// TIA Portal V15.1 export
// export: Created 2024-05-17T05:38:57.384126Z, ExportSetting WithDefaults, DisplayName Totally Integrated Automation Portal, DisplayVersion V15.1 Update 5, DisplayName TIA Portal Openness, DisplayVersion V15.1 Update 5, DisplayName SINAMICS Startdrive Advanced, DisplayVersion V15.1, DisplayName G130, G150, S120, S150, SINAMICS MV, S210, DisplayVersion V15.1, DisplayName G110M, G120, G120C, G120D, G120P, DisplayVersion V15.1, DisplayName STEP 7 Professional, DisplayVersion V15.1 Update 5, DisplayName STEP 7 Safety, DisplayVersion V15.1, DisplayName WinCC Professional, DisplayVersion V15.1 Update 5, DisplayName SIMATIC Visualization Architect, DisplayVersion V15.1
FUNCTION "209210ZS01Safety" : Void   // FC325, FBD
TITLE = 209210ZS01 Safety
{ S7_Optimized_Access := 'FALSE' }
AUTHOR : VCG
FAMILY : Local
NAME : 610
VERSION : 0.1
// stored: AutoNumber false, IsIECCheckEnabled false, SetENOAutomatically False, UDAEnableTagReadback false
   VAR_OUTPUT
      O_AlarmA : Bool;   // Alarm A
      O_AlarmB : Bool;   // Alarm B
      O_AlarmC : Bool;   // Alarm C
      O_AlarmD : Bool;   // Alarm D
      O_AlarmABCondition : Bool;   // Alarms resetable
      H_IAnim : Word;   // Icon Animation
   END_VAR
BEGIN

REGION Network 1: **** 2.1 - Enable Alarms **** 210CS22M4SG10F & SG11F Check if both safety sensors are activated
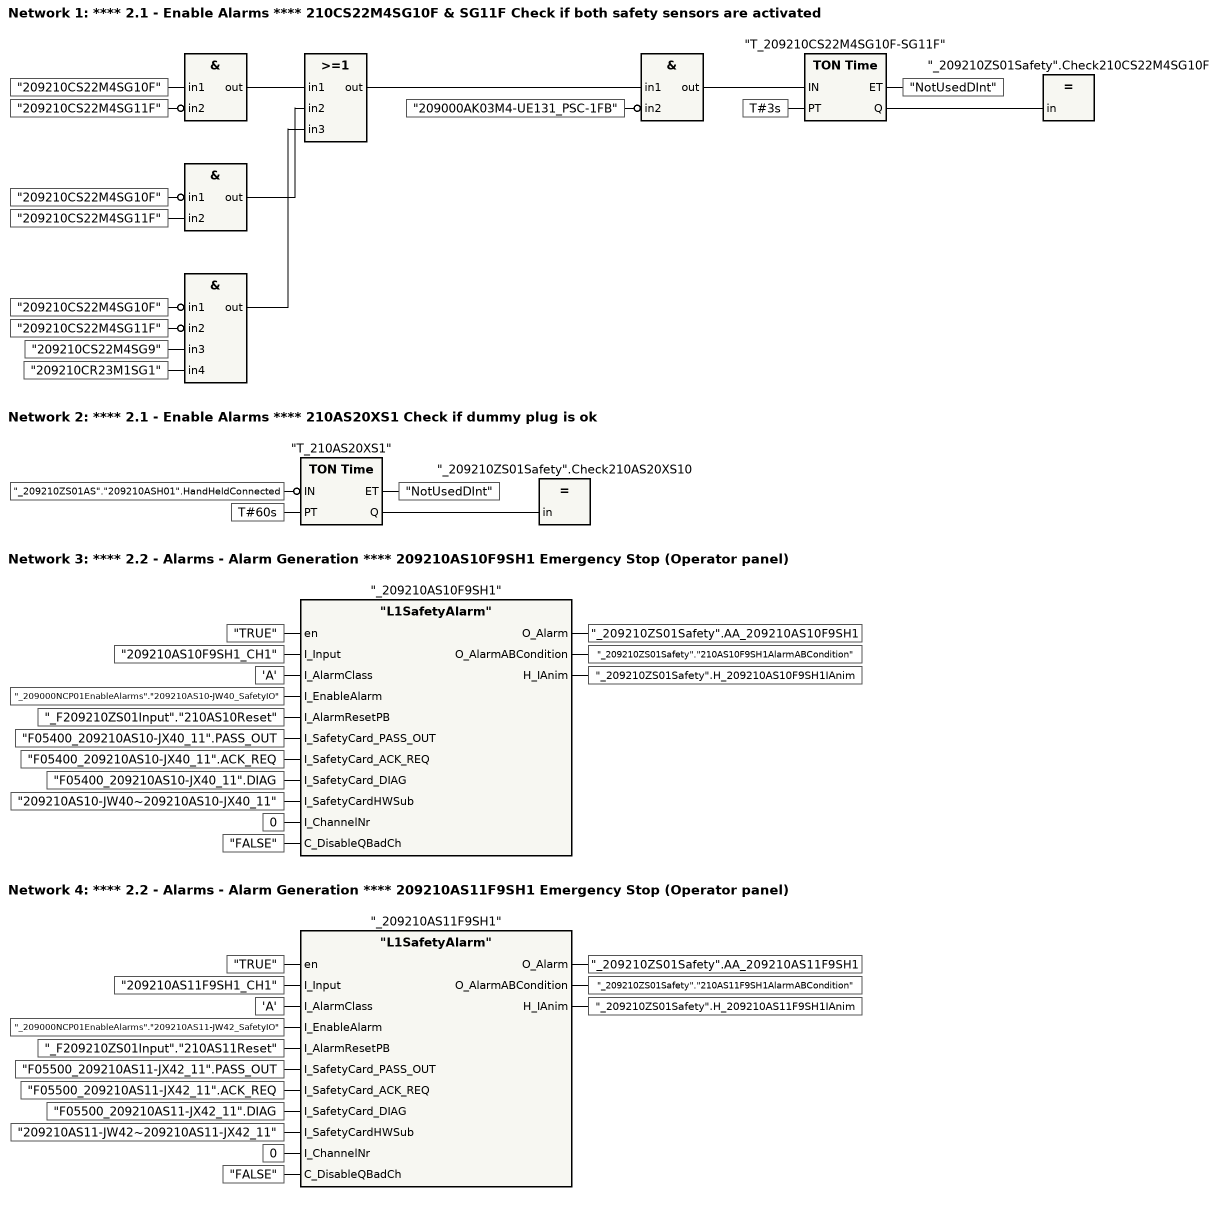
   "T_209210CS22M4SG10F-SG11F".TON(IN := (("209210CS22M4SG10F" AND NOT "209210CS22M4SG11F") OR (NOT "209210CS22M4SG10F" AND "209210CS22M4SG11F") OR (NOT "209210CS22M4SG10F" AND NOT "209210CS22M4SG11F" AND "209210CS22M4SG9" AND "209210CR23M1SG1")) AND NOT "209000AK03M4-UE131_PSC-1FB",
                           PT := T#3s,
                           ET => "NotUsedDInt");
   "_209210ZS01Safety".Check210CS22M4SG10F := "T_209210CS22M4SG10F-SG11F".Q;
END_REGION

REGION Network 2: **** 2.1 - Enable Alarms **** 210AS20XS1 Check if dummy plug is ok
   "T_210AS20XS1".TON(IN := NOT "_209210ZS01AS"."209210ASH01".HandHeldConnected,
                      PT := T#60s,
                      ET => "NotUsedDInt");
   "_209210ZS01Safety".Check210AS20XS10 := "T_210AS20XS1".Q;
END_REGION

REGION Network 3: **** 2.2 - Alarms - Alarm Generation **** 209210AS10F9SH1 Emergency Stop (Operator panel)
   // Emergency Stop
   IF "TRUE" THEN
       "_209210AS10F9SH1"(I_Input := "209210AS10F9SH1_CH1",   // "L1SafetyAlarm"
                          I_AlarmClass := 'A',
                          I_EnableAlarm := "_209000NCP01EnableAlarms"."209210AS10-JW40_SafetyIO",
                          I_AlarmResetPB := "_F209210ZS01Input"."210AS10Reset",
                          I_SafetyCard_PASS_OUT := "F05400_209210AS10-JX40_11".PASS_OUT,
                          I_SafetyCard_ACK_REQ := "F05400_209210AS10-JX40_11".ACK_REQ,
                          I_SafetyCard_DIAG := "F05400_209210AS10-JX40_11".DIAG,
                          I_SafetyCardHWSub := "209210AS10-JW40~209210AS10-JX40_11",
                          I_ChannelNr := 0,
                          C_DisableQBadCh := "FALSE",
                          O_Alarm => "_209210ZS01Safety".AA_209210AS10F9SH1,
                          O_AlarmABCondition => "_209210ZS01Safety"."210AS10F9SH1AlarmABCondition",
                          H_IAnim => "_209210ZS01Safety".H_209210AS10F9SH1IAnim);
   END_IF;
END_REGION

REGION Network 4: **** 2.2 - Alarms - Alarm Generation **** 209210AS11F9SH1 Emergency Stop (Operator panel)
   // Emergency Stop
   IF "TRUE" THEN
       "_209210AS11F9SH1"(I_Input := "209210AS11F9SH1_CH1",   // "L1SafetyAlarm"
                          I_AlarmClass := 'A',
                          I_EnableAlarm := "_209000NCP01EnableAlarms"."209210AS11-JW42_SafetyIO",
                          I_AlarmResetPB := "_F209210ZS01Input"."210AS11Reset",
                          I_SafetyCard_PASS_OUT := "F05500_209210AS11-JX42_11".PASS_OUT,
                          I_SafetyCard_ACK_REQ := "F05500_209210AS11-JX42_11".ACK_REQ,
                          I_SafetyCard_DIAG := "F05500_209210AS11-JX42_11".DIAG,
                          I_SafetyCardHWSub := "209210AS11-JW42~209210AS11-JX42_11",
                          I_ChannelNr := 0,
                          C_DisableQBadCh := "FALSE",
                          O_Alarm => "_209210ZS01Safety".AA_209210AS11F9SH1,
                          O_AlarmABCondition => "_209210ZS01Safety"."210AS11F9SH1AlarmABCondition",
                          H_IAnim => "_209210ZS01Safety".H_209210AS11F9SH1IAnim);
   END_IF;
END_REGION

REGION Network 5: **** 2.2 - Alarms - Alarm Generation **** 209210AS20F9SH1 Emergency Stop (Start/Stop panel)
   // Emergency Stop
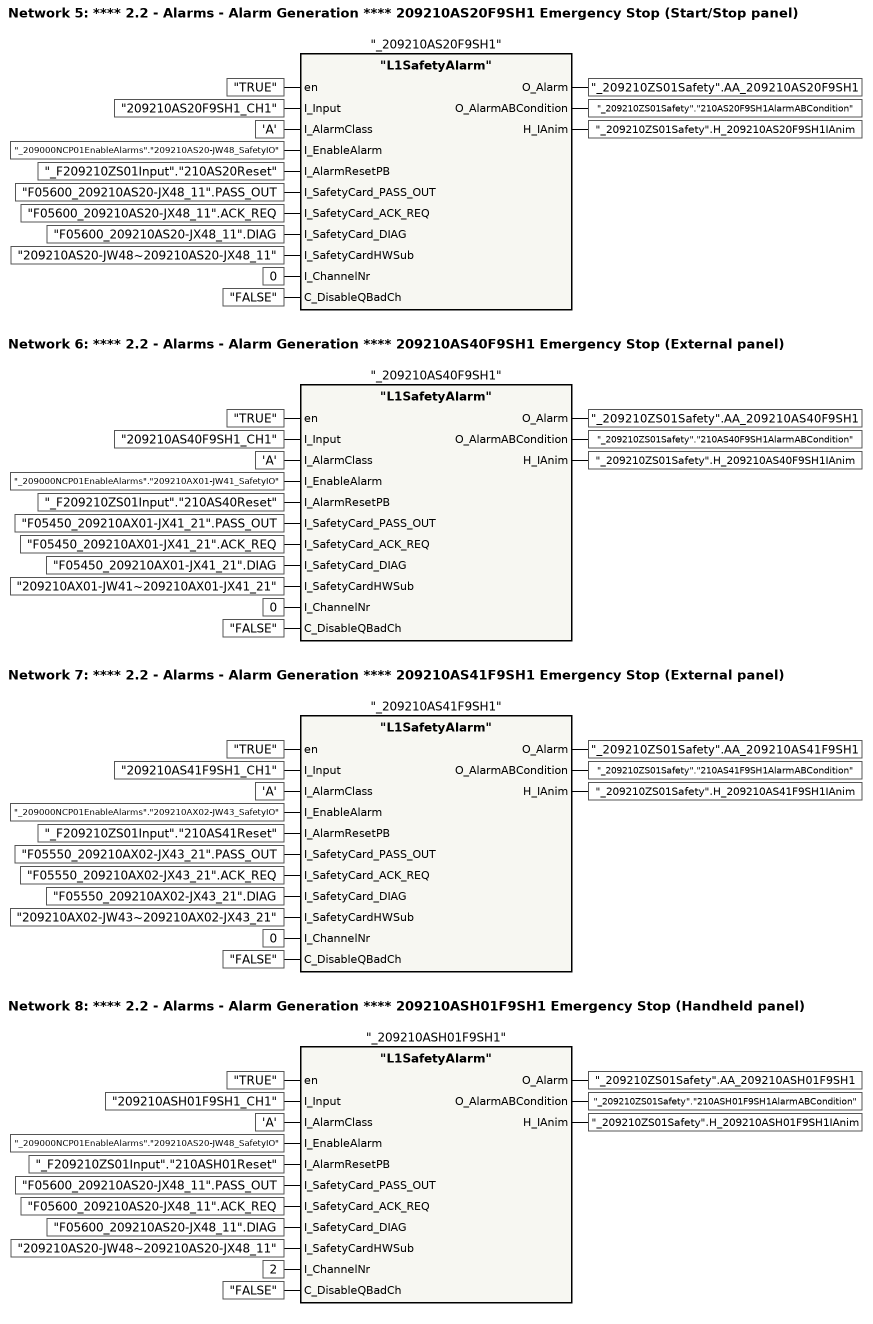
   IF "TRUE" THEN
       "_209210AS20F9SH1"(I_Input := "209210AS20F9SH1_CH1",   // "L1SafetyAlarm"
                          I_AlarmClass := 'A',
                          I_EnableAlarm := "_209000NCP01EnableAlarms"."209210AS20-JW48_SafetyIO",
                          I_AlarmResetPB := "_F209210ZS01Input"."210AS20Reset",
                          I_SafetyCard_PASS_OUT := "F05600_209210AS20-JX48_11".PASS_OUT,
                          I_SafetyCard_ACK_REQ := "F05600_209210AS20-JX48_11".ACK_REQ,
                          I_SafetyCard_DIAG := "F05600_209210AS20-JX48_11".DIAG,
                          I_SafetyCardHWSub := "209210AS20-JW48~209210AS20-JX48_11",
                          I_ChannelNr := 0,
                          C_DisableQBadCh := "FALSE",
                          O_Alarm => "_209210ZS01Safety".AA_209210AS20F9SH1,
                          O_AlarmABCondition => "_209210ZS01Safety"."210AS20F9SH1AlarmABCondition",
                          H_IAnim => "_209210ZS01Safety".H_209210AS20F9SH1IAnim);
   END_IF;
END_REGION

REGION Network 6: **** 2.2 - Alarms - Alarm Generation **** 209210AS40F9SH1 Emergency Stop (External panel)
   // Emergency Stop
   IF "TRUE" THEN
       "_209210AS40F9SH1"(I_Input := "209210AS40F9SH1_CH1",   // "L1SafetyAlarm"
                          I_AlarmClass := 'A',
                          I_EnableAlarm := "_209000NCP01EnableAlarms"."209210AX01-JW41_SafetyIO",
                          I_AlarmResetPB := "_F209210ZS01Input"."210AS40Reset",
                          I_SafetyCard_PASS_OUT := "F05450_209210AX01-JX41_21".PASS_OUT,
                          I_SafetyCard_ACK_REQ := "F05450_209210AX01-JX41_21".ACK_REQ,
                          I_SafetyCard_DIAG := "F05450_209210AX01-JX41_21".DIAG,
                          I_SafetyCardHWSub := "209210AX01-JW41~209210AX01-JX41_21",
                          I_ChannelNr := 0,
                          C_DisableQBadCh := "FALSE",
                          O_Alarm => "_209210ZS01Safety".AA_209210AS40F9SH1,
                          O_AlarmABCondition => "_209210ZS01Safety"."210AS40F9SH1AlarmABCondition",
                          H_IAnim => "_209210ZS01Safety".H_209210AS40F9SH1IAnim);
   END_IF;
END_REGION

REGION Network 7: **** 2.2 - Alarms - Alarm Generation **** 209210AS41F9SH1 Emergency Stop (External panel)
   // Emergency Stop
   IF "TRUE" THEN
       "_209210AS41F9SH1"(I_Input := "209210AS41F9SH1_CH1",   // "L1SafetyAlarm"
                          I_AlarmClass := 'A',
                          I_EnableAlarm := "_209000NCP01EnableAlarms"."209210AX02-JW43_SafetyIO",
                          I_AlarmResetPB := "_F209210ZS01Input"."210AS41Reset",
                          I_SafetyCard_PASS_OUT := "F05550_209210AX02-JX43_21".PASS_OUT,
                          I_SafetyCard_ACK_REQ := "F05550_209210AX02-JX43_21".ACK_REQ,
                          I_SafetyCard_DIAG := "F05550_209210AX02-JX43_21".DIAG,
                          I_SafetyCardHWSub := "209210AX02-JW43~209210AX02-JX43_21",
                          I_ChannelNr := 0,
                          C_DisableQBadCh := "FALSE",
                          O_Alarm => "_209210ZS01Safety".AA_209210AS41F9SH1,
                          O_AlarmABCondition => "_209210ZS01Safety"."210AS41F9SH1AlarmABCondition",
                          H_IAnim => "_209210ZS01Safety".H_209210AS41F9SH1IAnim);
   END_IF;
END_REGION

REGION Network 8: **** 2.2 - Alarms - Alarm Generation **** 209210ASH01F9SH1 Emergency Stop (Handheld panel)
   // Emergency Stop
   IF "TRUE" THEN
       "_209210ASH01F9SH1"(I_Input := "209210ASH01F9SH1_CH1",   // "L1SafetyAlarm"
                           I_AlarmClass := 'A',
                           I_EnableAlarm := "_209000NCP01EnableAlarms"."209210AS20-JW48_SafetyIO",
                           I_AlarmResetPB := "_F209210ZS01Input"."210ASH01Reset",
                           I_SafetyCard_PASS_OUT := "F05600_209210AS20-JX48_11".PASS_OUT,
                           I_SafetyCard_ACK_REQ := "F05600_209210AS20-JX48_11".ACK_REQ,
                           I_SafetyCard_DIAG := "F05600_209210AS20-JX48_11".DIAG,
                           I_SafetyCardHWSub := "209210AS20-JW48~209210AS20-JX48_11",
                           I_ChannelNr := 2,
                           C_DisableQBadCh := "FALSE",
                           O_Alarm => "_209210ZS01Safety".AA_209210ASH01F9SH1,
                           O_AlarmABCondition => "_209210ZS01Safety"."210ASH01F9SH1AlarmABCondition",
                           H_IAnim => "_209210ZS01Safety".H_209210ASH01F9SH1IAnim);
   END_IF;
END_REGION

REGION Network 9: **** 2.2 - Alarms - Alarm Generation **** 209210ASH01F9SH2 Deathmans switch (Handheld panel)
   // Deathmans switch
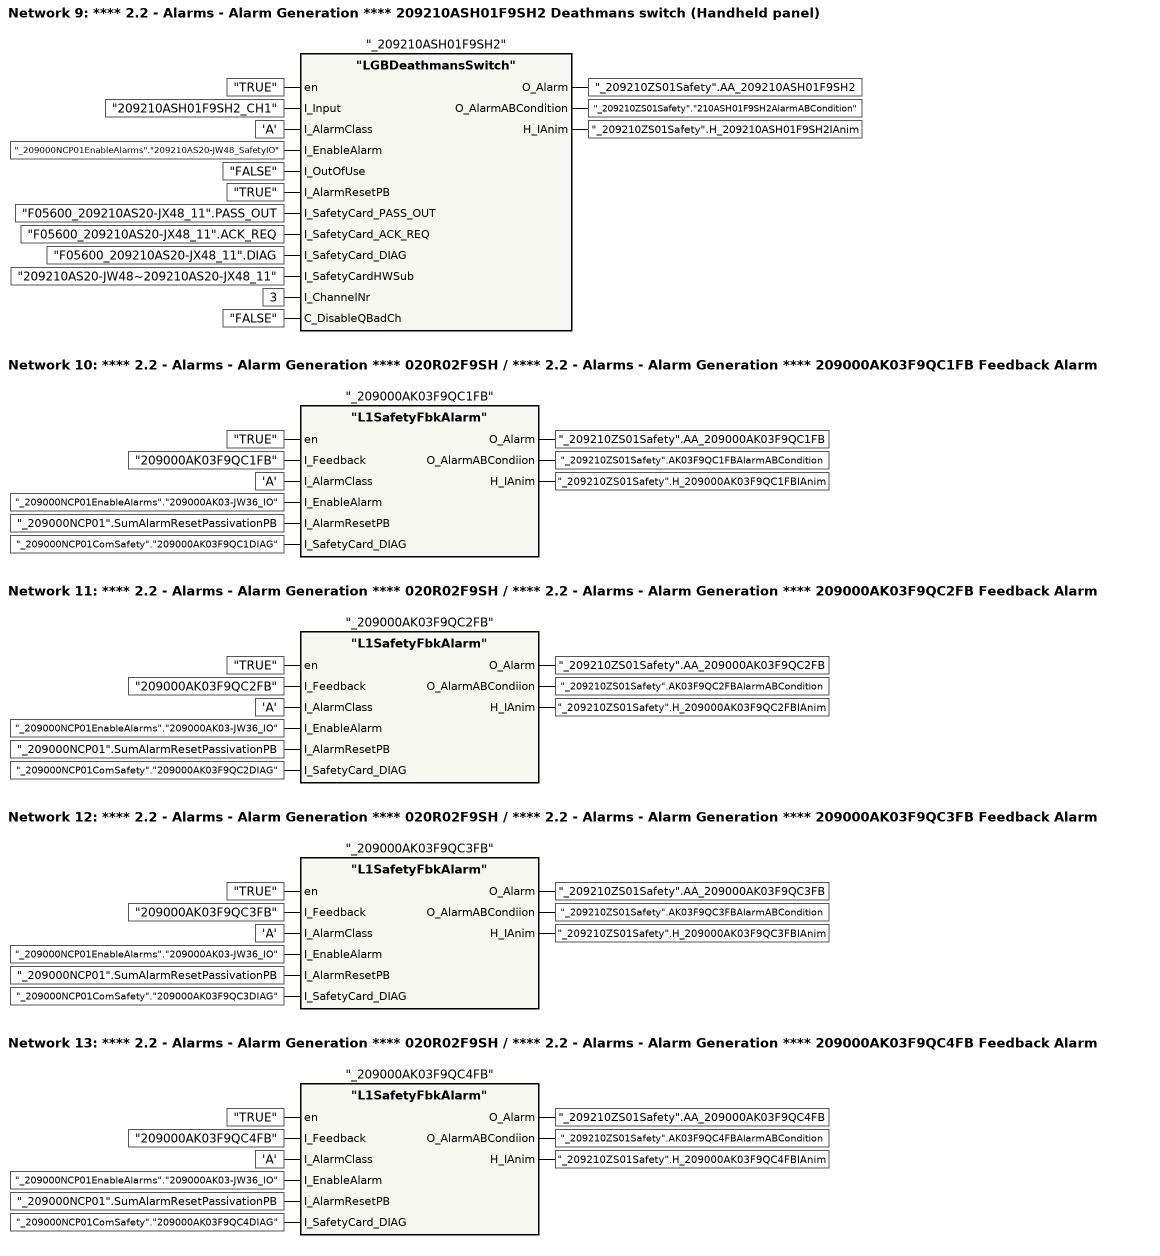
   IF "TRUE" THEN
       "_209210ASH01F9SH2"(I_Input := "209210ASH01F9SH2_CH1",   // "LGBDeathmansSwitch"
                           I_AlarmClass := 'A',
                           I_EnableAlarm := "_209000NCP01EnableAlarms"."209210AS20-JW48_SafetyIO",
                           I_OutOfUse := "FALSE",
                           I_AlarmResetPB := "TRUE",
                           I_SafetyCard_PASS_OUT := "F05600_209210AS20-JX48_11".PASS_OUT,
                           I_SafetyCard_ACK_REQ := "F05600_209210AS20-JX48_11".ACK_REQ,
                           I_SafetyCard_DIAG := "F05600_209210AS20-JX48_11".DIAG,
                           I_SafetyCardHWSub := "209210AS20-JW48~209210AS20-JX48_11",
                           I_ChannelNr := 3,
                           C_DisableQBadCh := "FALSE",
                           O_Alarm => "_209210ZS01Safety".AA_209210ASH01F9SH2,
                           O_AlarmABCondition => "_209210ZS01Safety"."210ASH01F9SH2AlarmABCondition",
                           H_IAnim => "_209210ZS01Safety".H_209210ASH01F9SH2IAnim);
   END_IF;
END_REGION

REGION Network 10: **** 2.2 - Alarms - Alarm Generation **** 020R02F9SH / **** 2.2 - Alarms - Alarm Generation **** 209000AK03F9QC1FB Feedback Alarm
   // E-Stop Push Button / Feedback Alarm
   IF "TRUE" THEN
       "_209000AK03F9QC1FB"(I_Feedback := "209000AK03F9QC1FB",   // "L1SafetyFbkAlarm"
                            I_AlarmClass := 'A',
                            I_EnableAlarm := "_209000NCP01EnableAlarms"."209000AK03-JW36_IO",
                            I_AlarmResetPB := "_209000NCP01".SumAlarmResetPassivationPB,
                            I_SafetyCard_DIAG := "_209000NCP01ComSafety"."209000AK03F9QC1DIAG",
                            O_Alarm => "_209210ZS01Safety".AA_209000AK03F9QC1FB,
                            O_AlarmABCondiion => "_209210ZS01Safety".AK03F9QC1FBAlarmABCondition,
                            H_IAnim => "_209210ZS01Safety".H_209000AK03F9QC1FBIAnim);
   END_IF;
END_REGION

REGION Network 11: **** 2.2 - Alarms - Alarm Generation **** 020R02F9SH / **** 2.2 - Alarms - Alarm Generation **** 209000AK03F9QC2FB Feedback Alarm
   // E-Stop Push Button / Feedback Alarm
   IF "TRUE" THEN
       "_209000AK03F9QC2FB"(I_Feedback := "209000AK03F9QC2FB",   // "L1SafetyFbkAlarm"
                            I_AlarmClass := 'A',
                            I_EnableAlarm := "_209000NCP01EnableAlarms"."209000AK03-JW36_IO",
                            I_AlarmResetPB := "_209000NCP01".SumAlarmResetPassivationPB,
                            I_SafetyCard_DIAG := "_209000NCP01ComSafety"."209000AK03F9QC2DIAG",
                            O_Alarm => "_209210ZS01Safety".AA_209000AK03F9QC2FB,
                            O_AlarmABCondiion => "_209210ZS01Safety".AK03F9QC2FBAlarmABCondition,
                            H_IAnim => "_209210ZS01Safety".H_209000AK03F9QC2FBIAnim);
   END_IF;
END_REGION

REGION Network 12: **** 2.2 - Alarms - Alarm Generation **** 020R02F9SH / **** 2.2 - Alarms - Alarm Generation **** 209000AK03F9QC3FB Feedback Alarm
   // E-Stop Push Button / Feedback Alarm
   IF "TRUE" THEN
       "_209000AK03F9QC3FB"(I_Feedback := "209000AK03F9QC3FB",   // "L1SafetyFbkAlarm"
                            I_AlarmClass := 'A',
                            I_EnableAlarm := "_209000NCP01EnableAlarms"."209000AK03-JW36_IO",
                            I_AlarmResetPB := "_209000NCP01".SumAlarmResetPassivationPB,
                            I_SafetyCard_DIAG := "_209000NCP01ComSafety"."209000AK03F9QC3DIAG",
                            O_Alarm => "_209210ZS01Safety".AA_209000AK03F9QC3FB,
                            O_AlarmABCondiion => "_209210ZS01Safety".AK03F9QC3FBAlarmABCondition,
                            H_IAnim => "_209210ZS01Safety".H_209000AK03F9QC3FBIAnim);
   END_IF;
END_REGION

REGION Network 13: **** 2.2 - Alarms - Alarm Generation **** 020R02F9SH / **** 2.2 - Alarms - Alarm Generation **** 209000AK03F9QC4FB Feedback Alarm
   // E-Stop Push Button / Feedback Alarm
   IF "TRUE" THEN
       "_209000AK03F9QC4FB"(I_Feedback := "209000AK03F9QC4FB",   // "L1SafetyFbkAlarm"
                            I_AlarmClass := 'A',
                            I_EnableAlarm := "_209000NCP01EnableAlarms"."209000AK03-JW36_IO",
                            I_AlarmResetPB := "_209000NCP01".SumAlarmResetPassivationPB,
                            I_SafetyCard_DIAG := "_209000NCP01ComSafety"."209000AK03F9QC4DIAG",
                            O_Alarm => "_209210ZS01Safety".AA_209000AK03F9QC4FB,
                            O_AlarmABCondiion => "_209210ZS01Safety".AK03F9QC4FBAlarmABCondition,
                            H_IAnim => "_209210ZS01Safety".H_209000AK03F9QC4FBIAnim);
   END_IF;
END_REGION

REGION Network 14: **** 2.2 - Alarms - Alarm Generation **** 020R02F9SH / **** 2.2 - Alarms - Alarm Generation **** 209000AK03F9QC5FB Feedback Alarm
   // E-Stop Push Button / Feedback Alarm
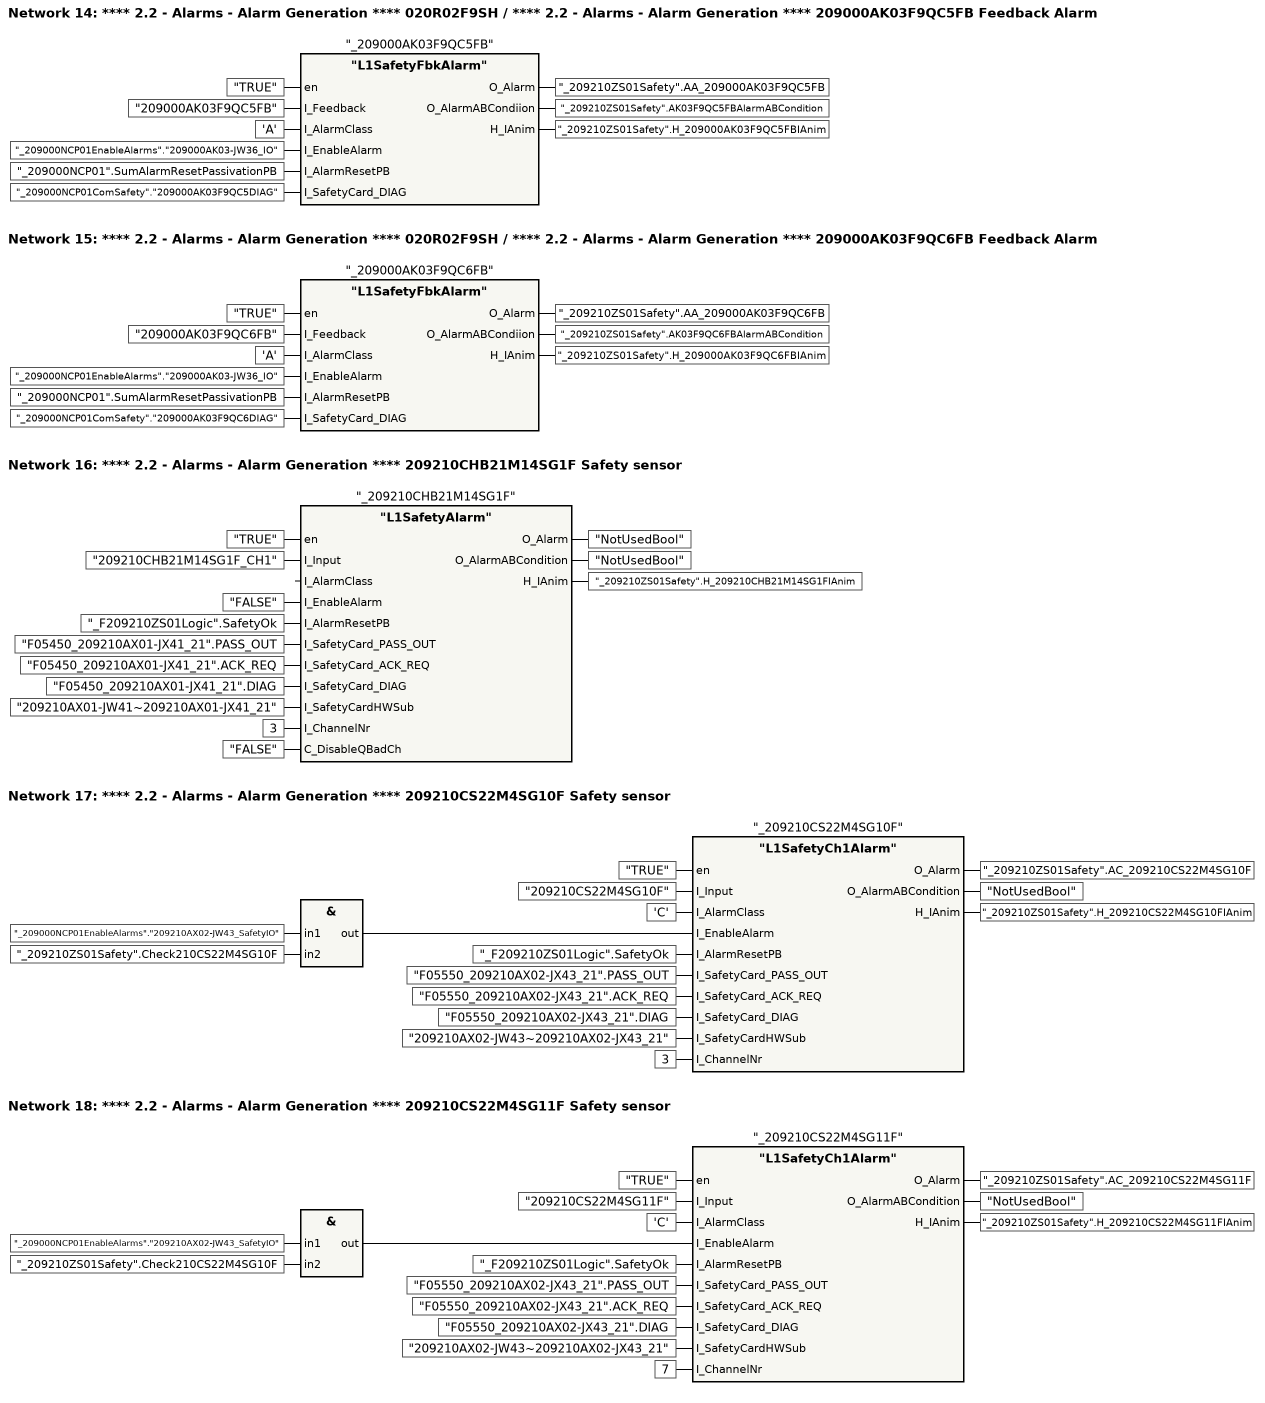
   IF "TRUE" THEN
       "_209000AK03F9QC5FB"(I_Feedback := "209000AK03F9QC5FB",   // "L1SafetyFbkAlarm"
                            I_AlarmClass := 'A',
                            I_EnableAlarm := "_209000NCP01EnableAlarms"."209000AK03-JW36_IO",
                            I_AlarmResetPB := "_209000NCP01".SumAlarmResetPassivationPB,
                            I_SafetyCard_DIAG := "_209000NCP01ComSafety"."209000AK03F9QC5DIAG",
                            O_Alarm => "_209210ZS01Safety".AA_209000AK03F9QC5FB,
                            O_AlarmABCondiion => "_209210ZS01Safety".AK03F9QC5FBAlarmABCondition,
                            H_IAnim => "_209210ZS01Safety".H_209000AK03F9QC5FBIAnim);
   END_IF;
END_REGION

REGION Network 15: **** 2.2 - Alarms - Alarm Generation **** 020R02F9SH / **** 2.2 - Alarms - Alarm Generation **** 209000AK03F9QC6FB Feedback Alarm
   // E-Stop Push Button / Feedback Alarm
   IF "TRUE" THEN
       "_209000AK03F9QC6FB"(I_Feedback := "209000AK03F9QC6FB",   // "L1SafetyFbkAlarm"
                            I_AlarmClass := 'A',
                            I_EnableAlarm := "_209000NCP01EnableAlarms"."209000AK03-JW36_IO",
                            I_AlarmResetPB := "_209000NCP01".SumAlarmResetPassivationPB,
                            I_SafetyCard_DIAG := "_209000NCP01ComSafety"."209000AK03F9QC6DIAG",
                            O_Alarm => "_209210ZS01Safety".AA_209000AK03F9QC6FB,
                            O_AlarmABCondiion => "_209210ZS01Safety".AK03F9QC6FBAlarmABCondition,
                            H_IAnim => "_209210ZS01Safety".H_209000AK03F9QC6FBIAnim);
   END_IF;
END_REGION

REGION Network 16: **** 2.2 - Alarms - Alarm Generation **** 209210CHB21M14SG1F Safety sensor
   // Safety sensor
   IF "TRUE" THEN
       "_209210CHB21M14SG1F"(I_Input := "209210CHB21M14SG1F_CH1",   // "L1SafetyAlarm"
                             I_EnableAlarm := "FALSE",
                             I_AlarmResetPB := "_F209210ZS01Logic".SafetyOk,
                             I_SafetyCard_PASS_OUT := "F05450_209210AX01-JX41_21".PASS_OUT,
                             I_SafetyCard_ACK_REQ := "F05450_209210AX01-JX41_21".ACK_REQ,
                             I_SafetyCard_DIAG := "F05450_209210AX01-JX41_21".DIAG,
                             I_SafetyCardHWSub := "209210AX01-JW41~209210AX01-JX41_21",
                             I_ChannelNr := 3,
                             C_DisableQBadCh := "FALSE",
                             O_Alarm => "NotUsedBool",
                             O_AlarmABCondition => "NotUsedBool",
                             H_IAnim => "_209210ZS01Safety".H_209210CHB21M14SG1FIAnim);
   END_IF;
END_REGION

REGION Network 17: **** 2.2 - Alarms - Alarm Generation **** 209210CS22M4SG10F Safety sensor
   // Safety sensor
   IF "TRUE" THEN
       "_209210CS22M4SG10F"(I_Input := "209210CS22M4SG10F",   // "L1SafetyCh1Alarm"
                            I_AlarmClass := 'C',
                            I_EnableAlarm := "_209000NCP01EnableAlarms"."209210AX02-JW43_SafetyIO" AND "_209210ZS01Safety".Check210CS22M4SG10F,
                            I_AlarmResetPB := "_F209210ZS01Logic".SafetyOk,
                            I_SafetyCard_PASS_OUT := "F05550_209210AX02-JX43_21".PASS_OUT,
                            I_SafetyCard_ACK_REQ := "F05550_209210AX02-JX43_21".ACK_REQ,
                            I_SafetyCard_DIAG := "F05550_209210AX02-JX43_21".DIAG,
                            I_SafetyCardHWSub := "209210AX02-JW43~209210AX02-JX43_21",
                            I_ChannelNr := 3,
                            O_Alarm => "_209210ZS01Safety".AC_209210CS22M4SG10F,
                            O_AlarmABCondition => "NotUsedBool",
                            H_IAnim => "_209210ZS01Safety".H_209210CS22M4SG10FIAnim);
   END_IF;
END_REGION

REGION Network 18: **** 2.2 - Alarms - Alarm Generation **** 209210CS22M4SG11F Safety sensor
   // Safety sensor
   IF "TRUE" THEN
       "_209210CS22M4SG11F"(I_Input := "209210CS22M4SG11F",   // "L1SafetyCh1Alarm"
                            I_AlarmClass := 'C',
                            I_EnableAlarm := "_209000NCP01EnableAlarms"."209210AX02-JW43_SafetyIO" AND "_209210ZS01Safety".Check210CS22M4SG10F,
                            I_AlarmResetPB := "_F209210ZS01Logic".SafetyOk,
                            I_SafetyCard_PASS_OUT := "F05550_209210AX02-JX43_21".PASS_OUT,
                            I_SafetyCard_ACK_REQ := "F05550_209210AX02-JX43_21".ACK_REQ,
                            I_SafetyCard_DIAG := "F05550_209210AX02-JX43_21".DIAG,
                            I_SafetyCardHWSub := "209210AX02-JW43~209210AX02-JX43_21",
                            I_ChannelNr := 7,
                            O_Alarm => "_209210ZS01Safety".AC_209210CS22M4SG11F,
                            O_AlarmABCondition => "NotUsedBool",
                            H_IAnim => "_209210ZS01Safety".H_209210CS22M4SG11FIAnim);
   END_IF;
END_REGION

REGION Network 19: **** 2.2 - Alarms - Alarm Generation **** 209210AS20XS10 Dummy plug
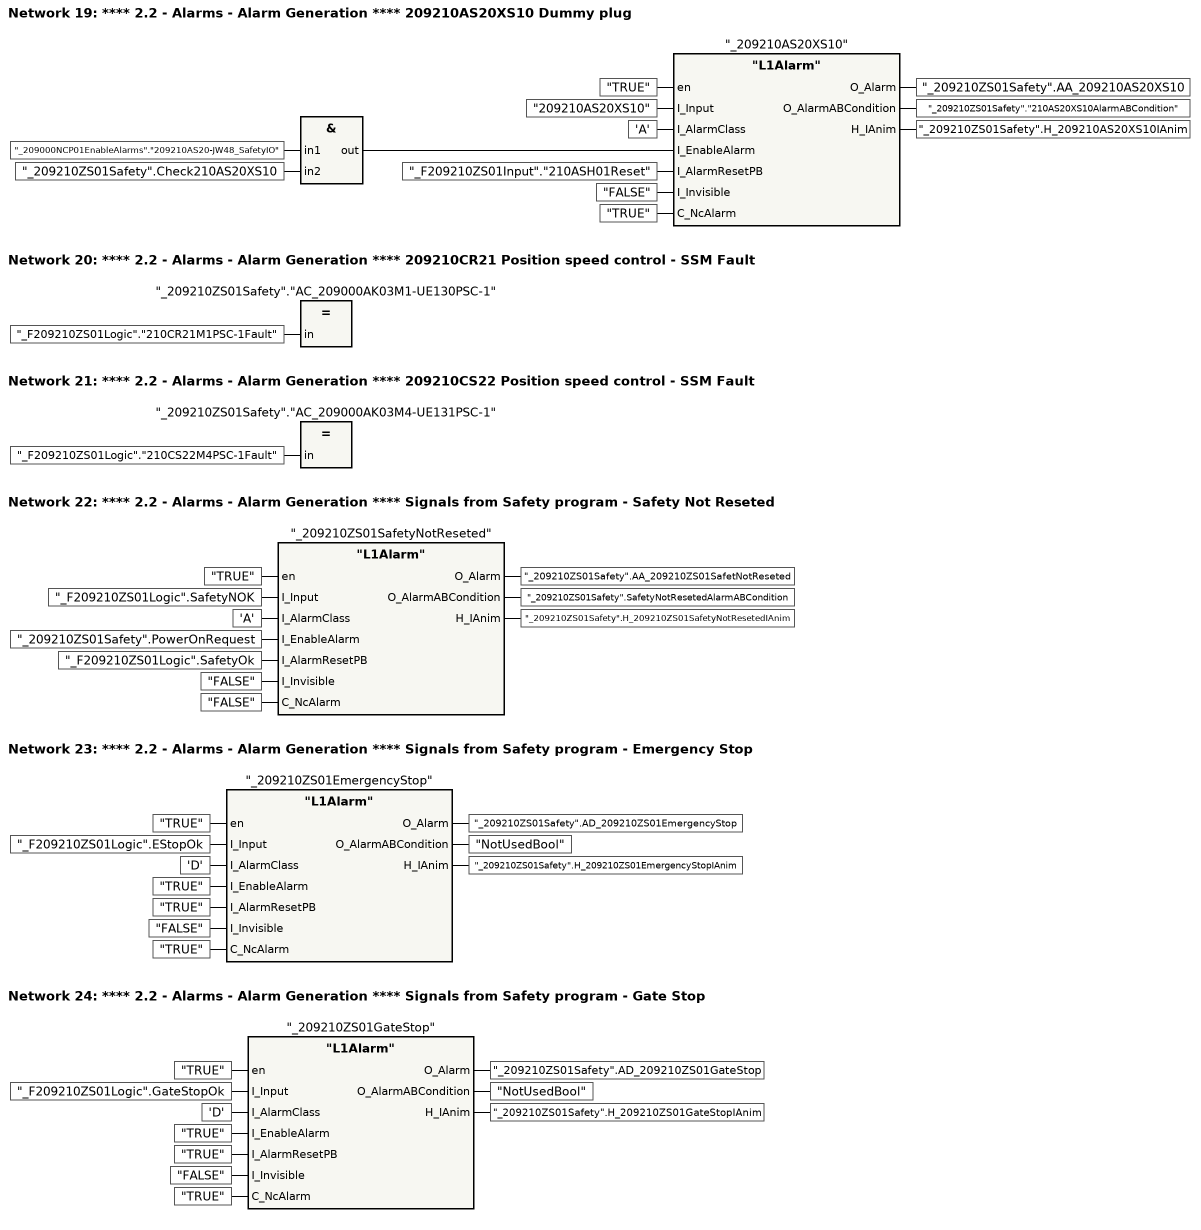
   IF "TRUE" THEN
       "_209210AS20XS10"(I_Input := "209210AS20XS10",   // "L1Alarm"
                         I_AlarmClass := 'A',
                         I_EnableAlarm := "_209000NCP01EnableAlarms"."209210AS20-JW48_SafetyIO" AND "_209210ZS01Safety".Check210AS20XS10,
                         I_AlarmResetPB := "_F209210ZS01Input"."210ASH01Reset",
                         I_Invisible := "FALSE",
                         C_NcAlarm := "TRUE",
                         O_Alarm => "_209210ZS01Safety".AA_209210AS20XS10,
                         O_AlarmABCondition => "_209210ZS01Safety"."210AS20XS10AlarmABCondition",
                         H_IAnim => "_209210ZS01Safety".H_209210AS20XS10IAnim);
   END_IF;
END_REGION

REGION Network 20: **** 2.2 - Alarms - Alarm Generation **** 209210CR21 Position speed control - SSM Fault
   // SEW Safety Function
   "_209210ZS01Safety"."AC_209000AK03M1-UE130PSC-1" := "_F209210ZS01Logic"."210CR21M1PSC-1Fault";
END_REGION

REGION Network 21: **** 2.2 - Alarms - Alarm Generation **** 209210CS22 Position speed control - SSM Fault
   // SEW Safety Function
   "_209210ZS01Safety"."AC_209000AK03M4-UE131PSC-1" := "_F209210ZS01Logic"."210CS22M4PSC-1Fault";
END_REGION

REGION Network 22: **** 2.2 - Alarms - Alarm Generation **** Signals from Safety program - Safety Not Reseted
   // Safety Has Not Been Reseted
   IF "TRUE" THEN
       "_209210ZS01SafetyNotReseted"(I_Input := "_F209210ZS01Logic".SafetyNOK,   // "L1Alarm"
                               I_AlarmClass := 'A',
                               I_EnableAlarm := "_209210ZS01Safety".PowerOnRequest,
                               I_AlarmResetPB := "_F209210ZS01Logic".SafetyOk,
                               I_Invisible := "FALSE",
                               C_NcAlarm := "FALSE",
                               O_Alarm => "_209210ZS01Safety".AA_209210ZS01SafetNotReseted,
                               O_AlarmABCondition => "_209210ZS01Safety".SafetyNotResetedAlarmABCondition,
                               H_IAnim => "_209210ZS01Safety".H_209210ZS01SafetyNotResetedIAnim);
   END_IF;
END_REGION

REGION Network 23: **** 2.2 - Alarms - Alarm Generation **** Signals from Safety program - Emergency Stop
   // Emergency Stop
   IF "TRUE" THEN
       "_209210ZS01EmergencyStop"(I_Input := "_F209210ZS01Logic".EStopOk,   // "L1Alarm"
                               I_AlarmClass := 'D',
                               I_EnableAlarm := "TRUE",
                               I_AlarmResetPB := "TRUE",
                               I_Invisible := "FALSE",
                               C_NcAlarm := "TRUE",
                               O_Alarm => "_209210ZS01Safety".AD_209210ZS01EmergencyStop,
                               O_AlarmABCondition => "NotUsedBool",
                               H_IAnim => "_209210ZS01Safety".H_209210ZS01EmergencyStopIAnim);
   END_IF;
END_REGION

REGION Network 24: **** 2.2 - Alarms - Alarm Generation **** Signals from Safety program - Gate Stop
   // Gate Stop
   IF "TRUE" THEN
       "_209210ZS01GateStop"(I_Input := "_F209210ZS01Logic".GateStopOk,   // "L1Alarm"
                             I_AlarmClass := 'D',
                             I_EnableAlarm := "TRUE",
                             I_AlarmResetPB := "TRUE",
                             I_Invisible := "FALSE",
                             C_NcAlarm := "TRUE",
                             O_Alarm => "_209210ZS01Safety".AD_209210ZS01GateStop,
                             O_AlarmABCondition => "NotUsedBool",
                             H_IAnim => "_209210ZS01Safety".H_209210ZS01GateStopIAnim);
   END_IF;
END_REGION

REGION Network 25: **** 2.2 - Alarms - Alarm Generation **** Signals from Safety program - Feedback Error
   // Feedback Error
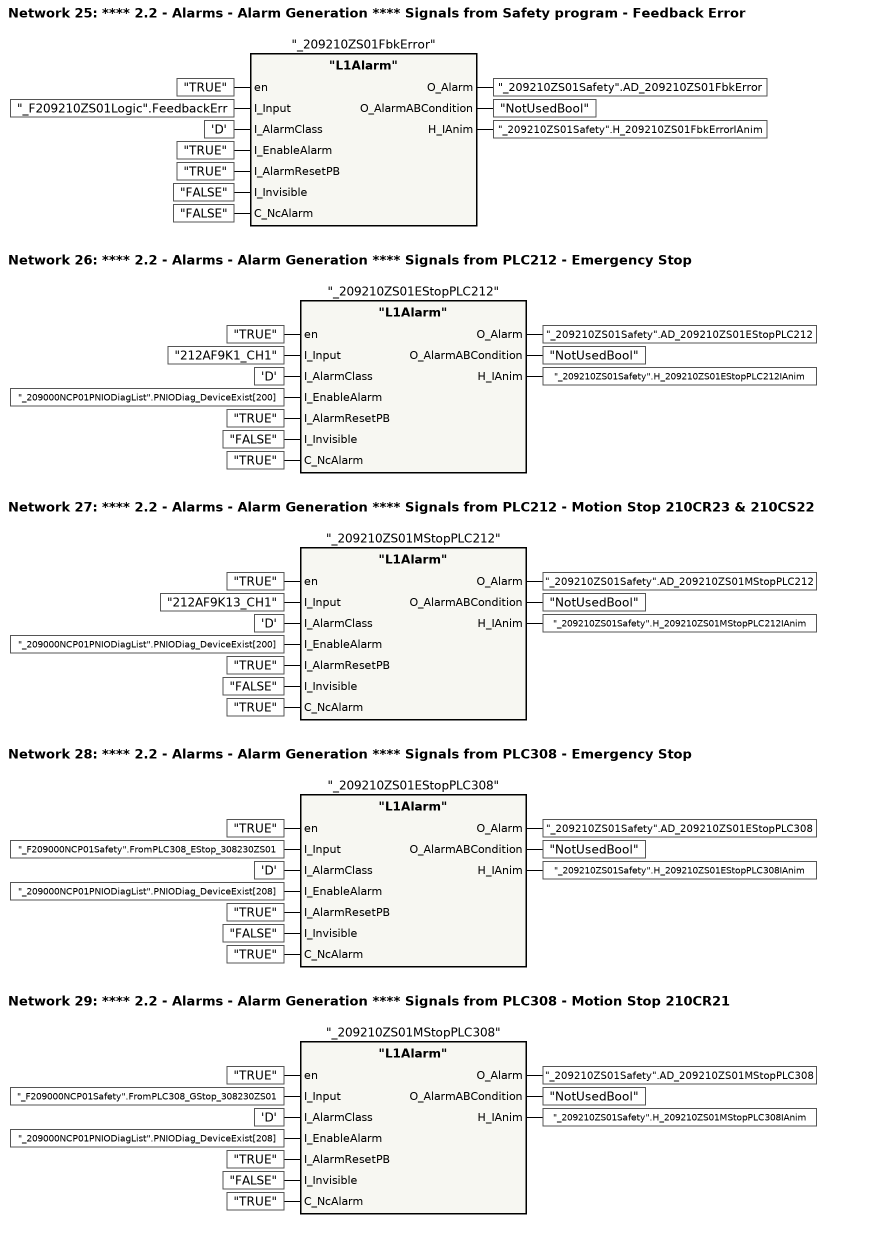
   IF "TRUE" THEN
       "_209210ZS01FbkError"(I_Input := "_F209210ZS01Logic".FeedbackErr,   // "L1Alarm"
                             I_AlarmClass := 'D',
                             I_EnableAlarm := "TRUE",
                             I_AlarmResetPB := "TRUE",
                             I_Invisible := "FALSE",
                             C_NcAlarm := "FALSE",
                             O_Alarm => "_209210ZS01Safety".AD_209210ZS01FbkError,
                             O_AlarmABCondition => "NotUsedBool",
                             H_IAnim => "_209210ZS01Safety".H_209210ZS01FbkErrorIAnim);
   END_IF;
END_REGION

REGION Network 26: **** 2.2 - Alarms - Alarm Generation **** Signals from PLC212 - Emergency Stop
   IF "TRUE" THEN
       "_209210ZS01EStopPLC212"(I_Input := "212AF9K1_CH1",   // "L1Alarm"
                               I_AlarmClass := 'D',
                               I_EnableAlarm := "_209000NCP01PNIODiagList".PNIODiag_DeviceExist[200],
                               I_AlarmResetPB := "TRUE",
                               I_Invisible := "FALSE",
                               C_NcAlarm := "TRUE",
                               O_Alarm => "_209210ZS01Safety".AD_209210ZS01EStopPLC212,
                               O_AlarmABCondition => "NotUsedBool",
                               H_IAnim => "_209210ZS01Safety".H_209210ZS01EStopPLC212IAnim);
   END_IF;
END_REGION

REGION Network 27: **** 2.2 - Alarms - Alarm Generation **** Signals from PLC212 - Motion Stop 210CR23 & 210CS22
   IF "TRUE" THEN
       "_209210ZS01MStopPLC212"(I_Input := "212AF9K13_CH1",   // "L1Alarm"
                               I_AlarmClass := 'D',
                               I_EnableAlarm := "_209000NCP01PNIODiagList".PNIODiag_DeviceExist[200],
                               I_AlarmResetPB := "TRUE",
                               I_Invisible := "FALSE",
                               C_NcAlarm := "TRUE",
                               O_Alarm => "_209210ZS01Safety".AD_209210ZS01MStopPLC212,
                               O_AlarmABCondition => "NotUsedBool",
                               H_IAnim => "_209210ZS01Safety".H_209210ZS01MStopPLC212IAnim);
   END_IF;
END_REGION

REGION Network 28: **** 2.2 - Alarms - Alarm Generation **** Signals from PLC308 - Emergency Stop
   IF "TRUE" THEN
       "_209210ZS01EStopPLC308"(I_Input := "_F209000NCP01Safety".FromPLC308_EStop_308230ZS01,   // "L1Alarm"
                               I_AlarmClass := 'D',
                               I_EnableAlarm := "_209000NCP01PNIODiagList".PNIODiag_DeviceExist[208],
                               I_AlarmResetPB := "TRUE",
                               I_Invisible := "FALSE",
                               C_NcAlarm := "TRUE",
                               O_Alarm => "_209210ZS01Safety".AD_209210ZS01EStopPLC308,
                               O_AlarmABCondition => "NotUsedBool",
                               H_IAnim => "_209210ZS01Safety".H_209210ZS01EStopPLC308IAnim);
   END_IF;
END_REGION

REGION Network 29: **** 2.2 - Alarms - Alarm Generation **** Signals from PLC308 - Motion Stop 210CR21
   IF "TRUE" THEN
       "_209210ZS01MStopPLC308"(I_Input := "_F209000NCP01Safety".FromPLC308_GStop_308230ZS01,   // "L1Alarm"
                               I_AlarmClass := 'D',
                               I_EnableAlarm := "_209000NCP01PNIODiagList".PNIODiag_DeviceExist[208],
                               I_AlarmResetPB := "TRUE",
                               I_Invisible := "FALSE",
                               C_NcAlarm := "TRUE",
                               O_Alarm => "_209210ZS01Safety".AD_209210ZS01MStopPLC308,
                               O_AlarmABCondition => "NotUsedBool",
                               H_IAnim => "_209210ZS01Safety".H_209210ZS01MStopPLC308IAnim);
   END_IF;
END_REGION

REGION Network 30: **** 3 - Communication - Devices **** Passivation
   // Passivation
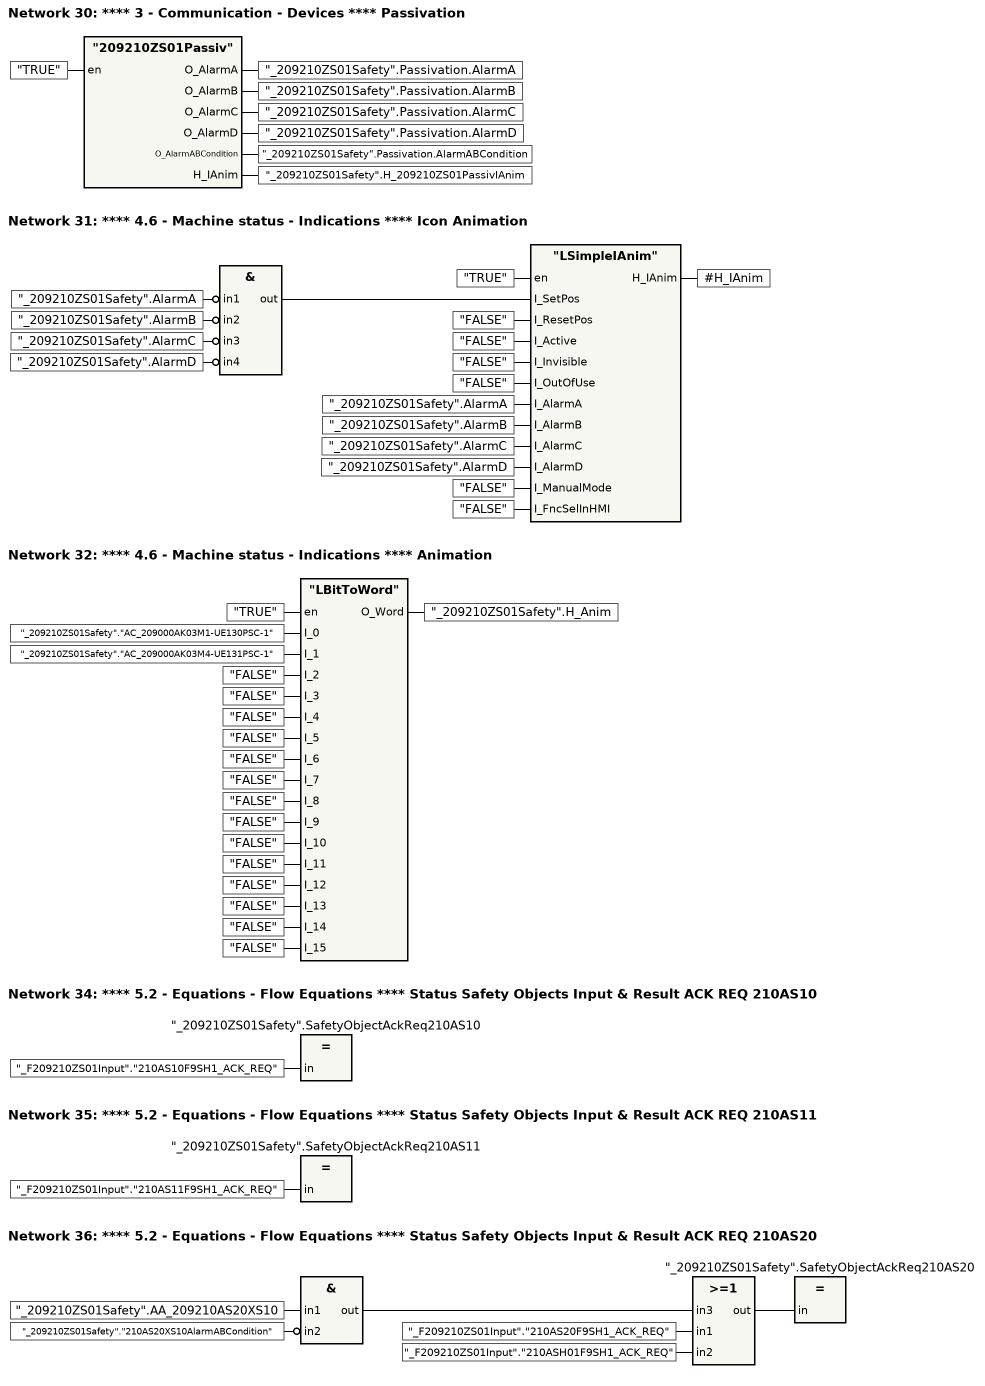
   IF "TRUE" THEN
       "209210ZS01Passiv"(O_AlarmA => "_209210ZS01Safety".Passivation.AlarmA,
                          O_AlarmB => "_209210ZS01Safety".Passivation.AlarmB,
                          O_AlarmC => "_209210ZS01Safety".Passivation.AlarmC,
                          O_AlarmD => "_209210ZS01Safety".Passivation.AlarmD,
                          O_AlarmABCondition => "_209210ZS01Safety".Passivation.AlarmABCondition,
                          H_IAnim => "_209210ZS01Safety".H_209210ZS01PassivIAnim);
   END_IF;
END_REGION

REGION Network 31: **** 4.6 - Machine status - Indications **** Icon Animation
   // Icon animation
   IF "TRUE" THEN
       "LSimpleIAnim"(I_SetPos := NOT "_209210ZS01Safety".AlarmA AND NOT "_209210ZS01Safety".AlarmB AND NOT "_209210ZS01Safety".AlarmC AND NOT "_209210ZS01Safety".AlarmD,
                      I_ResetPos := "FALSE",
                      I_Active := "FALSE",
                      I_Invisible := "FALSE",
                      I_OutOfUse := "FALSE",
                      I_AlarmA := "_209210ZS01Safety".AlarmA,
                      I_AlarmB := "_209210ZS01Safety".AlarmB,
                      I_AlarmC := "_209210ZS01Safety".AlarmC,
                      I_AlarmD := "_209210ZS01Safety".AlarmD,
                      I_ManualMode := "FALSE",
                      I_FncSelInHMI := "FALSE",
                      H_IAnim => #H_IAnim);
   END_IF;
END_REGION

REGION Network 32: **** 4.6 - Machine status - Indications **** Animation
   // Animation
   IF "TRUE" THEN
       "LBitToWord"(I_0 := "_209210ZS01Safety"."AC_209000AK03M1-UE130PSC-1",
                    I_1 := "_209210ZS01Safety"."AC_209000AK03M4-UE131PSC-1",
                    I_2 := "FALSE",
                    I_3 := "FALSE",
                    I_4 := "FALSE",
                    I_5 := "FALSE",
                    I_6 := "FALSE",
                    I_7 := "FALSE",
                    I_8 := "FALSE",
                    I_9 := "FALSE",
                    I_10 := "FALSE",
                    I_11 := "FALSE",
                    I_12 := "FALSE",
                    I_13 := "FALSE",
                    I_14 := "FALSE",
                    I_15 := "FALSE",
                    O_Word => "_209210ZS01Safety".H_Anim);
   END_IF;
END_REGION

NETWORK
TITLE = **** 4.6 - Machine Status - Indications **** Animation DB number
// DB number
      OPN   "_209210ZS01Safety";
      L     DBNO;
      T     "_209210ZS01Safety".H_DBnr;

REGION Network 34: **** 5.2 - Equations - Flow Equations **** Status Safety Objects Input & Result ACK REQ 210AS10
   "_209210ZS01Safety".SafetyObjectAckReq210AS10 := "_F209210ZS01Input"."210AS10F9SH1_ACK_REQ";
END_REGION

REGION Network 35: **** 5.2 - Equations - Flow Equations **** Status Safety Objects Input & Result ACK REQ 210AS11
   "_209210ZS01Safety".SafetyObjectAckReq210AS11 := "_F209210ZS01Input"."210AS11F9SH1_ACK_REQ";
END_REGION

REGION Network 36: **** 5.2 - Equations - Flow Equations **** Status Safety Objects Input & Result ACK REQ 210AS20
   "_209210ZS01Safety".SafetyObjectAckReq210AS20 := ("_209210ZS01Safety".AA_209210AS20XS10 AND NOT "_209210ZS01Safety"."210AS20XS10AlarmABCondition") OR "_F209210ZS01Input"."210AS20F9SH1_ACK_REQ" OR "_F209210ZS01Input"."210ASH01F9SH1_ACK_REQ";
END_REGION

REGION Network 37: **** 5.2 - Equations - Flow Equations **** Status Safety Objects Input & Result ACK REQ 210AS40
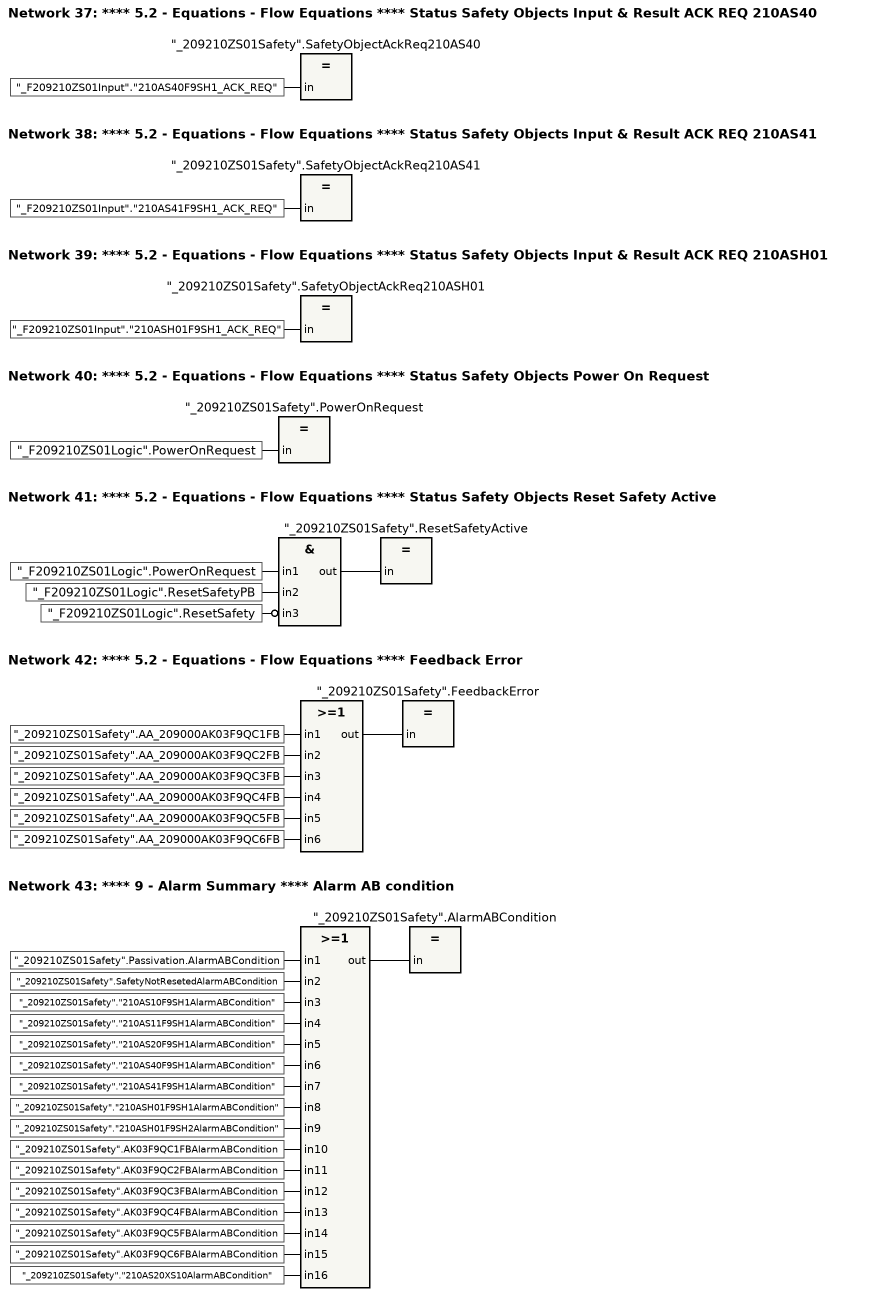
   "_209210ZS01Safety".SafetyObjectAckReq210AS40 := "_F209210ZS01Input"."210AS40F9SH1_ACK_REQ";
END_REGION

REGION Network 38: **** 5.2 - Equations - Flow Equations **** Status Safety Objects Input & Result ACK REQ 210AS41
   "_209210ZS01Safety".SafetyObjectAckReq210AS41 := "_F209210ZS01Input"."210AS41F9SH1_ACK_REQ";
END_REGION

REGION Network 39: **** 5.2 - Equations - Flow Equations **** Status Safety Objects Input & Result ACK REQ 210ASH01
   "_209210ZS01Safety".SafetyObjectAckReq210ASH01 := "_F209210ZS01Input"."210ASH01F9SH1_ACK_REQ";
END_REGION

REGION Network 40: **** 5.2 - Equations - Flow Equations **** Status Safety Objects Power On Request
   "_209210ZS01Safety".PowerOnRequest := "_F209210ZS01Logic".PowerOnRequest;
END_REGION

REGION Network 41: **** 5.2 - Equations - Flow Equations **** Status Safety Objects Reset Safety Active
   "_209210ZS01Safety".ResetSafetyActive := "_F209210ZS01Logic".PowerOnRequest AND "_F209210ZS01Logic".ResetSafetyPB AND NOT "_F209210ZS01Logic".ResetSafety;
END_REGION

REGION Network 42: **** 5.2 - Equations - Flow Equations **** Feedback Error
   "_209210ZS01Safety".FeedbackError := "_209210ZS01Safety".AA_209000AK03F9QC1FB OR "_209210ZS01Safety".AA_209000AK03F9QC2FB OR "_209210ZS01Safety".AA_209000AK03F9QC3FB OR "_209210ZS01Safety".AA_209000AK03F9QC4FB OR "_209210ZS01Safety".AA_209000AK03F9QC5FB OR "_209210ZS01Safety".AA_209000AK03F9QC6FB;
END_REGION

REGION Network 43: **** 9 - Alarm Summary **** Alarm AB condition
   // Alarm AB condition
   "_209210ZS01Safety".AlarmABCondition := "_209210ZS01Safety".Passivation.AlarmABCondition OR "_209210ZS01Safety".SafetyNotResetedAlarmABCondition OR "_209210ZS01Safety"."210AS10F9SH1AlarmABCondition" OR "_209210ZS01Safety"."210AS11F9SH1AlarmABCondition" OR "_209210ZS01Safety"."210AS20F9SH1AlarmABCondition" OR "_209210ZS01Safety"."210AS40F9SH1AlarmABCondition" OR "_209210ZS01Safety"."210AS41F9SH1AlarmABCondition" OR "_209210ZS01Safety"."210ASH01F9SH1AlarmABCondition" OR "_209210ZS01Safety"."210ASH01F9SH2AlarmABCondition" OR "_209210ZS01Safety".AK03F9QC1FBAlarmABCondition OR "_209210ZS01Safety".AK03F9QC2FBAlarmABCondition OR "_209210ZS01Safety".AK03F9QC3FBAlarmABCondition OR "_209210ZS01Safety".AK03F9QC4FBAlarmABCondition OR "_209210ZS01Safety".AK03F9QC5FBAlarmABCondition OR "_209210ZS01Safety".AK03F9QC6FBAlarmABCondition OR "_209210ZS01Safety"."210AS20XS10AlarmABCondition";
END_REGION

REGION Network 44: **** 9 - Alarm Summary **** Alarm A
   // Summary of alarms A
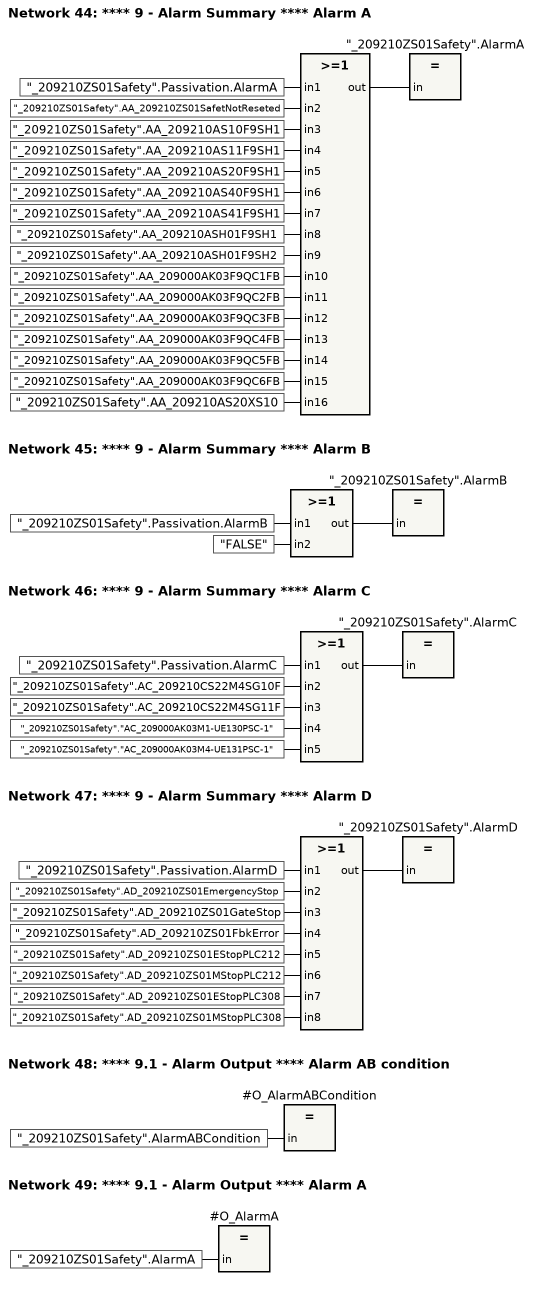
   "_209210ZS01Safety".AlarmA := "_209210ZS01Safety".Passivation.AlarmA OR "_209210ZS01Safety".AA_209210ZS01SafetNotReseted OR "_209210ZS01Safety".AA_209210AS10F9SH1 OR "_209210ZS01Safety".AA_209210AS11F9SH1 OR "_209210ZS01Safety".AA_209210AS20F9SH1 OR "_209210ZS01Safety".AA_209210AS40F9SH1 OR "_209210ZS01Safety".AA_209210AS41F9SH1 OR "_209210ZS01Safety".AA_209210ASH01F9SH1 OR "_209210ZS01Safety".AA_209210ASH01F9SH2 OR "_209210ZS01Safety".AA_209000AK03F9QC1FB OR "_209210ZS01Safety".AA_209000AK03F9QC2FB OR "_209210ZS01Safety".AA_209000AK03F9QC3FB OR "_209210ZS01Safety".AA_209000AK03F9QC4FB OR "_209210ZS01Safety".AA_209000AK03F9QC5FB OR "_209210ZS01Safety".AA_209000AK03F9QC6FB OR "_209210ZS01Safety".AA_209210AS20XS10;
END_REGION

REGION Network 45: **** 9 - Alarm Summary **** Alarm B
   // Summary of alarms B
   "_209210ZS01Safety".AlarmB := "_209210ZS01Safety".Passivation.AlarmB OR "FALSE";
END_REGION

REGION Network 46: **** 9 - Alarm Summary **** Alarm C
   // Summary of alarms C
   "_209210ZS01Safety".AlarmC := "_209210ZS01Safety".Passivation.AlarmC OR "_209210ZS01Safety".AC_209210CS22M4SG10F OR "_209210ZS01Safety".AC_209210CS22M4SG11F OR "_209210ZS01Safety"."AC_209000AK03M1-UE130PSC-1" OR "_209210ZS01Safety"."AC_209000AK03M4-UE131PSC-1";
END_REGION

REGION Network 47: **** 9 - Alarm Summary **** Alarm D
   // Summary of alarms D
   "_209210ZS01Safety".AlarmD := "_209210ZS01Safety".Passivation.AlarmD OR "_209210ZS01Safety".AD_209210ZS01EmergencyStop OR "_209210ZS01Safety".AD_209210ZS01GateStop OR "_209210ZS01Safety".AD_209210ZS01FbkError OR "_209210ZS01Safety".AD_209210ZS01EStopPLC212 OR "_209210ZS01Safety".AD_209210ZS01MStopPLC212 OR "_209210ZS01Safety".AD_209210ZS01EStopPLC308 OR "_209210ZS01Safety".AD_209210ZS01MStopPLC308;
END_REGION

REGION Network 48: **** 9.1 - Alarm Output **** Alarm AB condition
   // Alarm AB condition
   #O_AlarmABCondition := "_209210ZS01Safety".AlarmABCondition;
END_REGION

REGION Network 49: **** 9.1 - Alarm Output **** Alarm A
   // Summary of alarms A
   #O_AlarmA := "_209210ZS01Safety".AlarmA;
END_REGION

REGION Network 50: **** 9.1 - Alarm Output **** Alarm B
   // Summary of alarms B
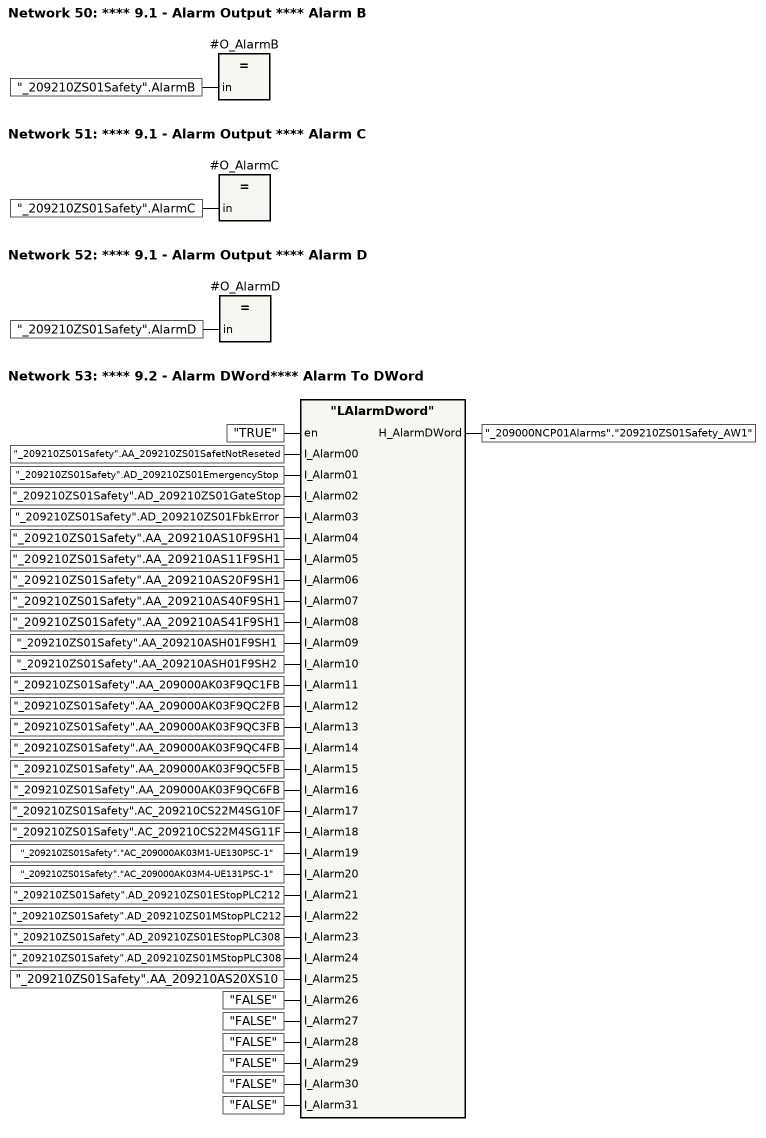
   #O_AlarmB := "_209210ZS01Safety".AlarmB;
END_REGION

REGION Network 51: **** 9.1 - Alarm Output **** Alarm C
   // Summary of alarms C
   #O_AlarmC := "_209210ZS01Safety".AlarmC;
END_REGION

REGION Network 52: **** 9.1 - Alarm Output **** Alarm D
   // Summary of alarms D
   #O_AlarmD := "_209210ZS01Safety".AlarmD;
END_REGION

REGION Network 53: **** 9.2 - Alarm DWord**** Alarm To DWord
   // Alarm Word
   IF "TRUE" THEN
       "LAlarmDword"(I_Alarm00 := "_209210ZS01Safety".AA_209210ZS01SafetNotReseted,
                     I_Alarm01 := "_209210ZS01Safety".AD_209210ZS01EmergencyStop,
                     I_Alarm02 := "_209210ZS01Safety".AD_209210ZS01GateStop,
                     I_Alarm03 := "_209210ZS01Safety".AD_209210ZS01FbkError,
                     I_Alarm04 := "_209210ZS01Safety".AA_209210AS10F9SH1,
                     I_Alarm05 := "_209210ZS01Safety".AA_209210AS11F9SH1,
                     I_Alarm06 := "_209210ZS01Safety".AA_209210AS20F9SH1,
                     I_Alarm07 := "_209210ZS01Safety".AA_209210AS40F9SH1,
                     I_Alarm08 := "_209210ZS01Safety".AA_209210AS41F9SH1,
                     I_Alarm09 := "_209210ZS01Safety".AA_209210ASH01F9SH1,
                     I_Alarm10 := "_209210ZS01Safety".AA_209210ASH01F9SH2,
                     I_Alarm11 := "_209210ZS01Safety".AA_209000AK03F9QC1FB,
                     I_Alarm12 := "_209210ZS01Safety".AA_209000AK03F9QC2FB,
                     I_Alarm13 := "_209210ZS01Safety".AA_209000AK03F9QC3FB,
                     I_Alarm14 := "_209210ZS01Safety".AA_209000AK03F9QC4FB,
                     I_Alarm15 := "_209210ZS01Safety".AA_209000AK03F9QC5FB,
                     I_Alarm16 := "_209210ZS01Safety".AA_209000AK03F9QC6FB,
                     I_Alarm17 := "_209210ZS01Safety".AC_209210CS22M4SG10F,
                     I_Alarm18 := "_209210ZS01Safety".AC_209210CS22M4SG11F,
                     I_Alarm19 := "_209210ZS01Safety"."AC_209000AK03M1-UE130PSC-1",
                     I_Alarm20 := "_209210ZS01Safety"."AC_209000AK03M4-UE131PSC-1",
                     I_Alarm21 := "_209210ZS01Safety".AD_209210ZS01EStopPLC212,
                     I_Alarm22 := "_209210ZS01Safety".AD_209210ZS01MStopPLC212,
                     I_Alarm23 := "_209210ZS01Safety".AD_209210ZS01EStopPLC308,
                     I_Alarm24 := "_209210ZS01Safety".AD_209210ZS01MStopPLC308,
                     I_Alarm25 := "_209210ZS01Safety".AA_209210AS20XS10,
                     I_Alarm26 := "FALSE",
                     I_Alarm27 := "FALSE",
                     I_Alarm28 := "FALSE",
                     I_Alarm29 := "FALSE",
                     I_Alarm30 := "FALSE",
                     I_Alarm31 := "FALSE",
                     H_AlarmDWord => "_209000NCP01Alarms"."209210ZS01Safety_AW1");
   END_IF;
END_REGION
END_FUNCTION
